{attribute 'qualified_only'}
VAR_GLOBAL
	stJoystickX : ST_JoystickScale;
	stJoystickY : ST_JoystickScale; 
	stInputs : ST_InputScaling;
	stFlows : ST_FlowScale;
END_VAR

(* stored: Version 1.1.0.1, ProductVersion 3.1.4024.12
   GVL G_StructData: Id {022b2ed1-56b6-4316-9a28-558bbcaea34e} *)
